SUBAPPLICATION Uebung_089a_AX (* Beispiel für E_RF_TRIG, mit Plug and Socket *)
  (* Standard: 61499-2; Description: Copyright (c) 2026 Meisterschulen am Ostbahnhof This program and the accompanying materials are made available under the terms of the Eclipse Public License 2.0 which is available at https://www.eclipse.org/legal/epl-2.0/ SPDX-License-Identifier: EPL-2.0 *)
  (* Version 1.0, 2026-09-10, Franz Höpfinger, Meisterschulen am Ostbahnhof, initial API and implementation and/or initial documentation *)
  PACKAGE Uebungen;
  IMPORT logiBUS::io::DI::logiBUS_DI::Input_I1;
  IMPORT logiBUS::io::DQ::logiBUS_DO::Output_Q1;
  IMPORT logiBUS::io::DQ::logiBUS_DO::Output_Q2;
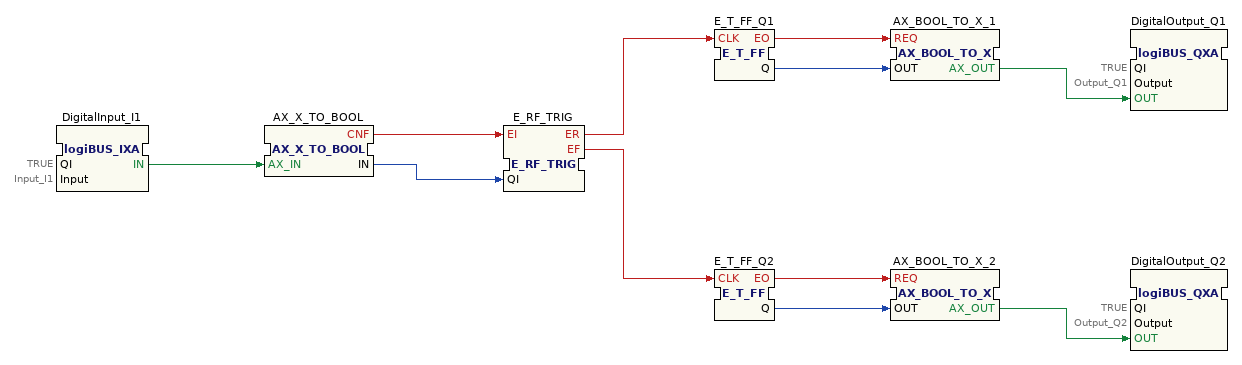
  (* Ein einziger Eingang, EIN Signal - E_RF_TRIG liefert beide Flanken gleichzeitig (ER=steigend, EF=fallend). Q1 togglet bei steigender, Q2 bei fallender Flanke. *)
  FBS
    DigitalInput_I1 : logiBUS::io::DI::logiBUS_IXA(QI := TRUE, Input := Input_I1);
    E_RF_TRIG : iec61499::events::E_RF_TRIG;
    E_T_FF_Q1 : iec61499::events::E_T_FF;
    E_T_FF_Q2 : iec61499::events::E_T_FF;
    DigitalOutput_Q1 : logiBUS::io::DQ::logiBUS_QXA(QI := TRUE, Output := Output_Q1);
    DigitalOutput_Q2 : logiBUS::io::DQ::logiBUS_QXA(QI := TRUE, Output := Output_Q2);
    AX_X_TO_BOOL : adapter::conversion::unidirectional::AX_X_TO_BOOL;
    AX_BOOL_TO_X_1 : adapter::conversion::unidirectional::AX_BOOL_TO_X;
    AX_BOOL_TO_X_2 : adapter::conversion::unidirectional::AX_BOOL_TO_X;
  END_FBS
  EVENT_CONNECTIONS
    AX_X_TO_BOOL.CNF TO E_RF_TRIG.EI;
    E_RF_TRIG.ER TO E_T_FF_Q1.CLK;
    E_RF_TRIG.EF TO E_T_FF_Q2.CLK;
    E_T_FF_Q1.EO TO AX_BOOL_TO_X_1.REQ;
    E_T_FF_Q2.EO TO AX_BOOL_TO_X_2.REQ;
  END_CONNECTIONS
  DATA_CONNECTIONS
    AX_X_TO_BOOL.IN TO E_RF_TRIG.QI;
    E_T_FF_Q1.Q TO AX_BOOL_TO_X_1.OUT;
    E_T_FF_Q2.Q TO AX_BOOL_TO_X_2.OUT;
  END_CONNECTIONS
  ADAPTER_CONNECTIONS
    DigitalInput_I1.IN TO AX_X_TO_BOOL.AX_IN;
    AX_BOOL_TO_X_1.AX_OUT TO DigitalOutput_Q1.OUT;
    AX_BOOL_TO_X_2.AX_OUT TO DigitalOutput_Q2.OUT;
  END_CONNECTIONS
END_SUBAPPLICATION
